{attribute 'qualified_only'}
{attribute 'strict'}
TYPE RFID_Error :
(
	None := 0,
	Not_Connected := 1,
	Time_Out := 2,
	Sesnor := 3
) UINT;
END_TYPE

(* stored: Version 1.1.0.1, ProductVersion 3.1.4024.10
   DUT RFID_Error: Id {1de2253f-3b50-4935-af52-71e4af814a2b} *)
